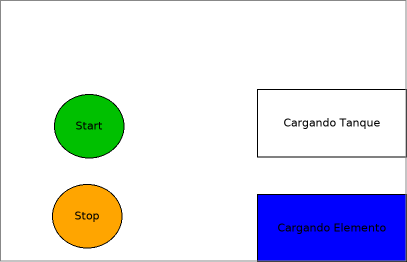
VISUALIZATION pantallaHMi  // 407x262
    Ellipse (54,94 70x64), "Start"
        toggle GVLvars.Start_Button
    Ellipse (52,184 70x64), "Stop"
        toggle GVLvars.StopButton
    RoundedRectangle (257,89 150x68), "Cargando Tanque"
        toggle GVLvars.Fill_Valve
    RoundedRectangle (257,194 150x68), "Cargando Elemento"
        toggle GVLvars.Discharge_Valve
END_VISUALIZATION

(* stored: Version 1.1.0.1, ProductVersion 3.1.4024.15
   Visu pantallaHMi: Id {24edfe00-072a-494b-8c89-3530fcfd886b} *)
